{attribute 'GeneratedUsingTerminal: ELM9410-0000-0016'}
{attribute addProperty BoxType "ELM9410-0000-0016"}
{attribute addProperty Id "Up_Out_OFFBOOL1"}
{attribute addProperty CRC "3958230902"}
{attribute addProperty Size "1"}
TYPE Control_EBEDCF76 :
STRUCT
	{attribute addProperty Name "Up_Out_OFF"}
	Up_Out_OFF : BOOL;
END_STRUCT
END_TYPE

(* stored: Version 1.2.0.0, ProductVersion 3.1.4024.9
   DUT Control_EBEDCF76: Id {47eedf2c-3281-4030-aa6a-394fd17e6fd8} *)
